(* Schneider Machine Expert - Basic project MIXER_EPP_STARTUP, file version 2.8.0.0 *)
(* CompanyInformations: Name=PROMASS, PhoneNumber=+39074238501, Street=Via XXV Aprile, 10/12, City=Trevi, ZipCode=06039, State=PG, Country=Italy, WebSite=www.promass.com *)
(* ProjectInformations: Name=MIXER_EPP, Description=CONTROL TO MIX-UP RECYCLED EPP (EXANDED POLYPROPILENE) WITH FRESH EPP.
AN ADDITIONAL BLOWE IS ADDED TO PERMIT THE OUTPUT FLOW *)
(* UserInformations: LastName=Torroni, FirstName=Stefano, PhoneNumber=+390742385051, Email=info@promass.com *)

HARDWARE
  Cpu 0: TM221CE16T
  EthernetConfiguration: NetworkName=M221, IpAllocationMode=FixedAddress, IpAddress=192.168.250.10, SubnetMask=255.255.255.0
  SerialLineConfiguration: Baud=Baud19200, Parity=ParityEven, DataBits=DataBits8, StopBits=StopBits1, PhysicalMedium=PhysicalMediumRs485, TransmissionMode=TransmissionModeIoScannerRtu
  MastTask: UsePeriodScanMode=false, PeriodScan=100
  FastTask: Period=255
  CpuBehavior: StartingMode=StartAutoRunForced, AutoSaveRamOnEeprom=true, WatchdogPeriod=250

SYMBOLS  (address, symbol, comment, settings)
  %M0       DRV_PWR_ON
  %M1       DRV0_JOG_INC
  %M2       DRV0_JOG_DEC
  %M3       DRV1_JOG_INC
  %M4       DRV1_JOG_DEC
  %M5       DRV0_MOVE_VEL
  %M6       DRV1_MOVE_VEL
  %M7       DRV0_ERROR
  %M8       DRV1_ERROR
  %M11      UPP_SENS_ON
  %M12      REM_TANK_FULL_V
  %M13      BLOWER_TOF
  %M100     RATIO_0_CHANGED
  %M101     RATIO_1_CHANGED
  %MW0      DRV0_JOG_SPEED
  %MW1      DRV1_JOG_SPEED
  %MW2      DRV0_MOVEVEL_SPEED
  %MW3      DRV1_MOVE_VEL_SPEED
  %MW4      HMI_ALARMS
  %MW5      FSM
  %MW6      HMI_INP  "HMI>>PLC COMMANDS"
  %MW7      HMI_OUT_00  "PLC>>HMI FEEDBACK WORD 01"
  %MW8      HMI_OUT_01  "PLC>>HMI FEEDBACK WORD 02"
  %MW9      SCREW_0_RATIO
  %MW10     SCREW_1_RATIO
  %MW11     BLOWER_DELAY_OFF
  %MW12     UPP_SENS_DELAY_ON
  %MW13     REM_TANK_SENS_DELAY_ON
  %TM11       [Type=TOF, Base=OneSecond, IsDynamicPreset=true]
  %TM13       [Base=OneSecond, IsDynamicPreset=true]
  %MC_JOG_ATV0   [Axis(Value(DriveAxis=DRV0)), Vel(Value(short=30))]
  %MC_JOG_ATV1   [Axis(Value(DriveAxis=DRV1)), Vel(Value(short=15))]
  %MC_MOVEVEL_ATV0   [Axis(Value(DriveAxis=DRV0)), Vel(Value(short=0))]
  %MC_MOVEVEL_ATV1   [Axis(Value(DriveAxis=DRV1)), Vel(Value(short=0))]
  %MC_POWER_ATV0   [Axis(Value(DriveAxis=DRV0))]
  %MC_POWER_ATV1   [Axis(Value(DriveAxis=DRV1))]
  %MC_READMOTIONSTATE_ATV0   [Axis(Value(DriveAxis=DRV0))]
  %MC_READMOTIONSTATE_ATV1   [Axis(Value(DriveAxis=DRV1))]
  %MC_READSTATUS_ATV0   [Axis(Value(DriveAxis=DRV0))]
  %MC_READSTATUS_ATV1   [Axis(Value(DriveAxis=DRV1))]
  %MC_RESET_ATV0   [Axis(Value(DriveAxis=DRV0))]
  %MC_RESET_ATV1   [Axis(Value(DriveAxis=DRV1))]
  %MC_STOP_ATV0   [Axis(Value(DriveAxis=DRV0))]
  %MC_STOP_ATV1   [Axis(Value(DriveAxis=DRV1))]
  %I0.0     START_BTN
  %I0.1     STOP_BTN
  %I0.2     I02
  %I0.3     QM1
  %I0.4     QM2
  %I0.5     QM3
  %I0.6     SK3
  %I0.7     MAT_LVL_UP
  %I0.8     REM_TANK_FULL
  %Q0.0     BLOWER

POU MAIN
  (* SectionNumber=1 *)

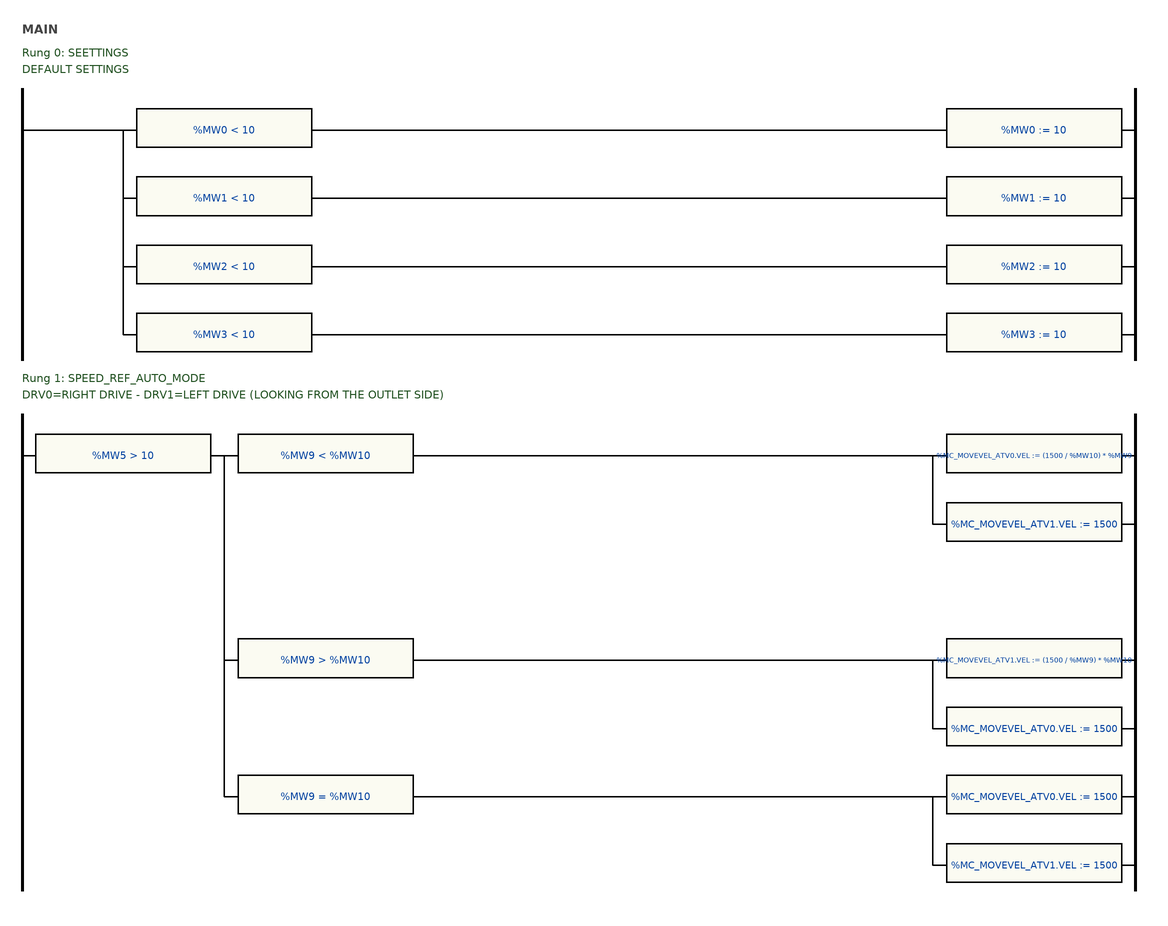

// Rung 0: SEETTINGS
// DEFAULT SETTINGS
  LD 1
  MPS
  AND [ %MW0 < 10 ]       (* DRV0_JOG_SPEED *)
  [ %MW0 := 10 ]          (* DRV0_JOG_SPEED *)
  MRD
  AND [ %MW1 < 10 ]       (* DRV1_JOG_SPEED *)
  [ %MW1 := 10 ]          (* DRV1_JOG_SPEED *)
  MRD
  AND [ %MW2 < 10 ]       (* DRV0_MOVEVEL_SPEED *)
  [ %MW2 := 10 ]          (* DRV0_MOVEVEL_SPEED *)
  MPP
  AND [ %MW3 < 10 ]       (* DRV1_MOVE_VEL_SPEED *)
  [ %MW3 := 10 ]          (* DRV1_MOVE_VEL_SPEED *)
  // as ST:
  //   IF DRV0_JOG_SPEED < 10 THEN DRV0_JOG_SPEED := 10; END_IF;
  //   IF DRV1_JOG_SPEED < 10 THEN DRV1_JOG_SPEED := 10; END_IF;
  //   IF DRV0_MOVEVEL_SPEED < 10 THEN DRV0_MOVEVEL_SPEED := 10; END_IF;
  //   IF DRV1_MOVE_VEL_SPEED < 10 THEN DRV1_MOVE_VEL_SPEED := 10; END_IF;

// Rung 1: SPEED_REF_AUTO_MODE
// DRV0=RIGHT DRIVE - DRV1=LEFT DRIVE (LOOKING FROM THE OUTLET SIDE)
  LD [ %MW5 > 10 ]        (* FSM *)
  MPS
  AND [ %MW9 < %MW10 ]    (* SCREW_0_RATIO, SCREW_1_RATIO *)
  [ %MC_MOVEVEL_ATV0.VEL := ( 1500 / %MW10 ) * %MW9 ](* SCREW_1_RATIO, SCREW_0_RATIO *)
  [ %MC_MOVEVEL_ATV1.VEL := 1500 ]
  MRD
  AND [ %MW9 > %MW10 ]    (* SCREW_0_RATIO, SCREW_1_RATIO *)
  [ %MC_MOVEVEL_ATV1.VEL := ( 1500 / %MW9 ) * %MW10 ](* SCREW_0_RATIO, SCREW_1_RATIO *)
  [ %MC_MOVEVEL_ATV0.VEL := 1500 ]
  MPP
  AND [ %MW9 = %MW10 ]    (* SCREW_0_RATIO, SCREW_1_RATIO *)
  [ %MC_MOVEVEL_ATV0.VEL := 1500 ]
  [ %MC_MOVEVEL_ATV1.VEL := 1500 ]
  // as ST:
  //   IF FSM > 10 AND SCREW_0_RATIO < SCREW_1_RATIO THEN %MC_MOVEVEL_ATV0.VEL := ( 1500 / SCREW_1_RATIO ) * SCREW_0_RATIO; END_IF;
  //   IF FSM > 10 AND SCREW_0_RATIO < SCREW_1_RATIO THEN %MC_MOVEVEL_ATV1.VEL := 1500; END_IF;
  //   IF FSM > 10 AND SCREW_0_RATIO > SCREW_1_RATIO THEN %MC_MOVEVEL_ATV1.VEL := ( 1500 / SCREW_0_RATIO ) * SCREW_1_RATIO; END_IF;
  //   IF FSM > 10 AND SCREW_0_RATIO > SCREW_1_RATIO THEN %MC_MOVEVEL_ATV0.VEL := 1500; END_IF;
  //   IF FSM > 10 AND SCREW_0_RATIO = SCREW_1_RATIO THEN %MC_MOVEVEL_ATV0.VEL := 1500; END_IF;
  //   IF FSM > 10 AND SCREW_0_RATIO = SCREW_1_RATIO THEN %MC_MOVEVEL_ATV1.VEL := 1500; END_IF;

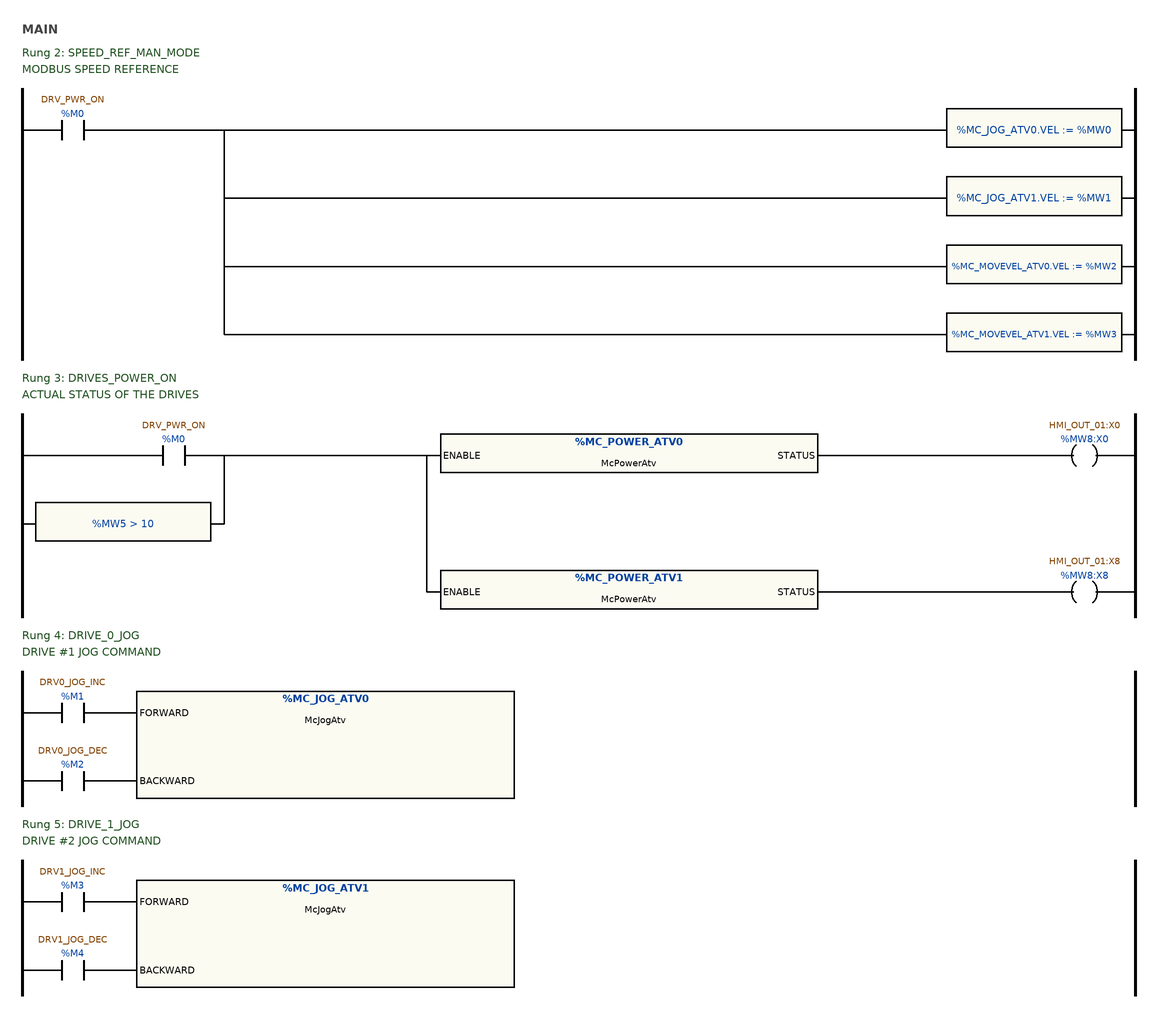

// Rung 2: SPEED_REF_MAN_MODE
// MODBUS SPEED REFERENCE
  LD %M0                  (* DRV_PWR_ON *)
  [ %MC_JOG_ATV0.VEL := %MW0 ](* DRV0_JOG_SPEED *)
  [ %MC_JOG_ATV1.VEL := %MW1 ](* DRV1_JOG_SPEED *)
  [ %MC_MOVEVEL_ATV0.VEL := %MW2 ](* DRV0_MOVEVEL_SPEED *)
  [ %MC_MOVEVEL_ATV1.VEL := %MW3 ](* DRV1_MOVE_VEL_SPEED *)
  // as ST:
  //   IF DRV_PWR_ON THEN %MC_JOG_ATV0.VEL := DRV0_JOG_SPEED; END_IF;
  //   IF DRV_PWR_ON THEN %MC_JOG_ATV1.VEL := DRV1_JOG_SPEED; END_IF;
  //   IF DRV_PWR_ON THEN %MC_MOVEVEL_ATV0.VEL := DRV0_MOVEVEL_SPEED; END_IF;
  //   IF DRV_PWR_ON THEN %MC_MOVEVEL_ATV1.VEL := DRV1_MOVE_VEL_SPEED; END_IF;

// Rung 3: DRIVES_POWER_ON
// ACTUAL STATUS OF THE DRIVES
  LD 1
  MULTIFB
  LD 1
  AND %M0                 (* DRV_PWR_ON *)
  OR [ %MW5 > 10 ]        (* FSM *)
  ST %MW2009:X0
  BLK %MC_POWER_ATV0
  LD %MW2009:X0
  ENABLE
  OUT_BLK
  LD STATUS
  ST %MW8:X0              (* HMI_OUT_01 *)
  END_BLK
  BLK %MC_POWER_ATV1
  LD %MW2009:X0
  ENABLE
  OUT_BLK
  LD STATUS
  ST %MW8:X8              (* HMI_OUT_01 *)
  END_BLK
  MULTIFB
  // as ST:
  //   %MC_POWER_ATV0(ENABLE := DRV_PWR_ON OR FSM > 10);
  //   HMI_OUT_01:X0 := %MC_POWER_ATV0.STATUS;
  //   %MC_POWER_ATV1(ENABLE := DRV_PWR_ON OR FSM > 10);
  //   HMI_OUT_01:X8 := %MC_POWER_ATV1.STATUS;

// Rung 4: DRIVE_0_JOG
// DRIVE #1 JOG COMMAND
  BLK %MC_JOG_ATV0
  LD %M1                  (* DRV0_JOG_INC *)
  FORWARD
  LD %M2                  (* DRV0_JOG_DEC *)
  BACKWARD
  END_BLK
  // as ST:
  //   %MC_JOG_ATV0(FORWARD := DRV0_JOG_INC, BACKWARD := DRV0_JOG_DEC);

// Rung 5: DRIVE_1_JOG
// DRIVE #2 JOG COMMAND
  BLK %MC_JOG_ATV1
  LD %M3                  (* DRV1_JOG_INC *)
  FORWARD
  LD %M4                  (* DRV1_JOG_DEC *)
  BACKWARD
  END_BLK
  // as ST:
  //   %MC_JOG_ATV1(FORWARD := DRV1_JOG_INC, BACKWARD := DRV1_JOG_DEC);

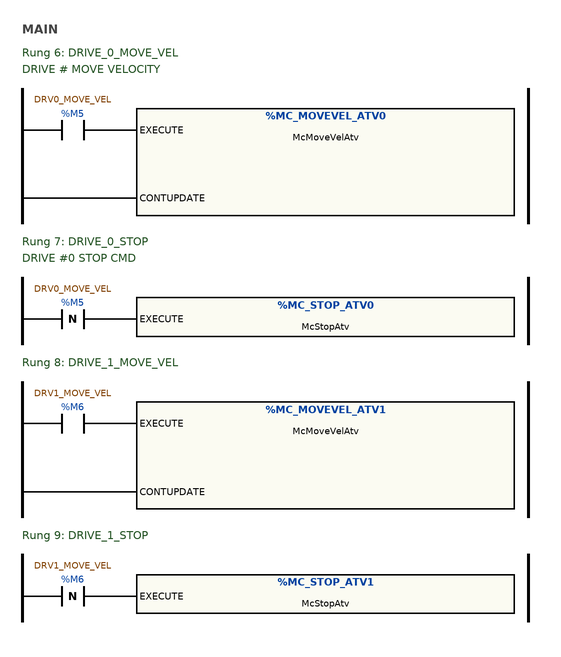

// Rung 6: DRIVE_0_MOVE_VEL
// DRIVE # MOVE VELOCITY
  BLK %MC_MOVEVEL_ATV0
  LD %M5                  (* DRV0_MOVE_VEL *)
  EXECUTE
  LD 1
  CONTUPDATE
  END_BLK
  // as ST:
  //   %MC_MOVEVEL_ATV0(EXECUTE := DRV0_MOVE_VEL, CONTUPDATE := TRUE);

// Rung 7: DRIVE_0_STOP
// DRIVE #0 STOP CMD
  BLK %MC_STOP_ATV0
  LDF %M5                 (* DRV0_MOVE_VEL *)
  EXECUTE
  END_BLK
  // as ST:
  //   %MC_STOP_ATV0(EXECUTE := FALLING(DRV0_MOVE_VEL));

// Rung 8: DRIVE_1_MOVE_VEL
  BLK %MC_MOVEVEL_ATV1
  LD %M6                  (* DRV1_MOVE_VEL *)
  EXECUTE
  LD 1
  CONTUPDATE
  END_BLK
  // as ST:
  //   %MC_MOVEVEL_ATV1(EXECUTE := DRV1_MOVE_VEL, CONTUPDATE := TRUE);

// Rung 9: DRIVE_1_STOP
  BLK %MC_STOP_ATV1
  LDF %M6                 (* DRV1_MOVE_VEL *)
  EXECUTE
  END_BLK
  // as ST:
  //   %MC_STOP_ATV1(EXECUTE := FALLING(DRV1_MOVE_VEL));

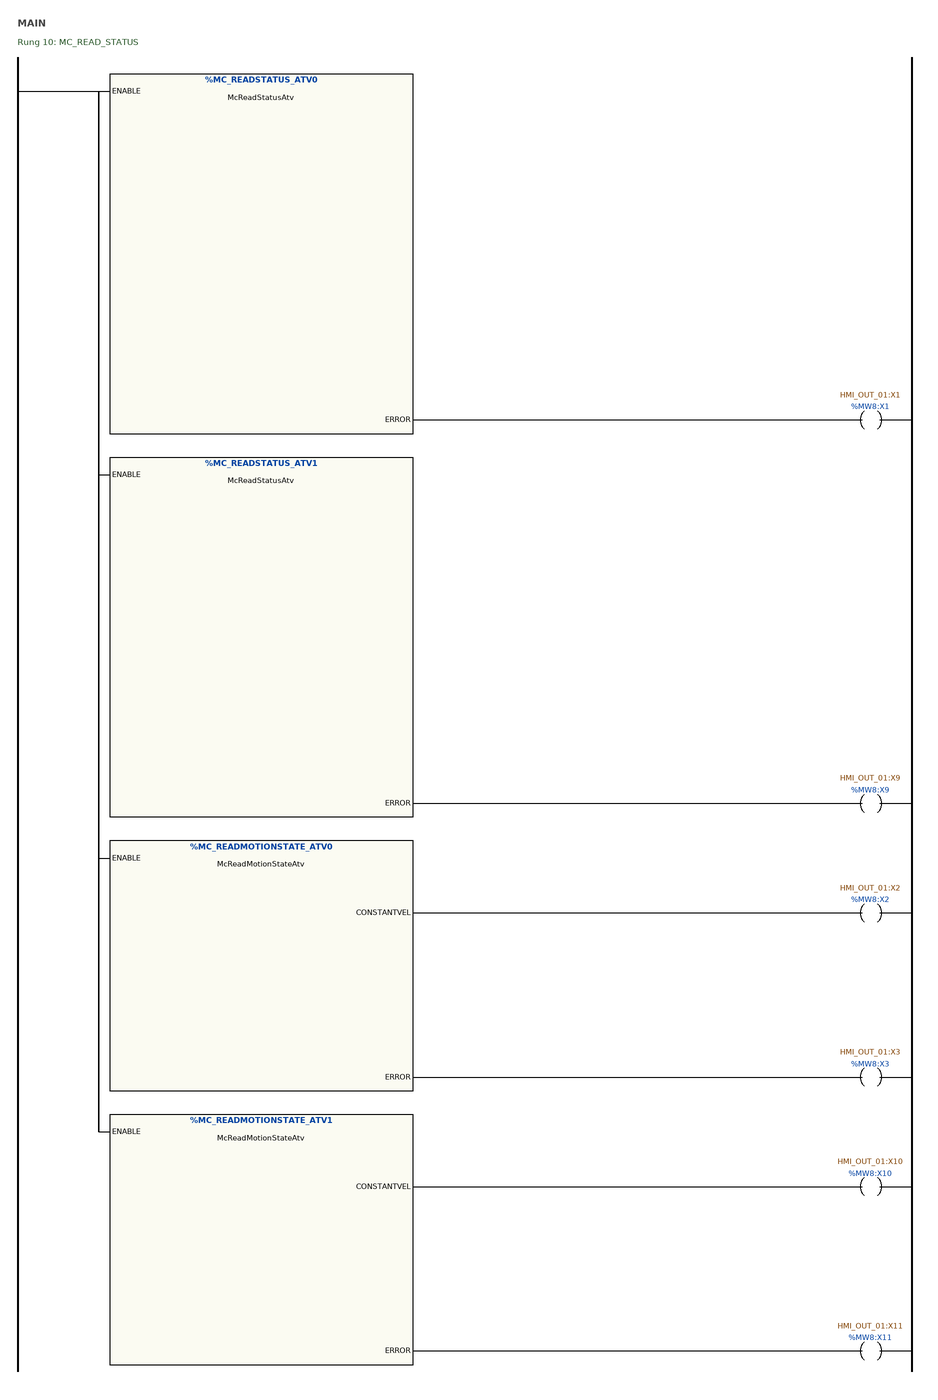

// Rung 10: MC_READ_STATUS
  LD 1
  MULTIFB
  LD 1
  ST %MW2009:X0
  BLK %MC_READSTATUS_ATV0
  LD %MW2009:X0
  ENABLE
  OUT_BLK
  LD ERROR
  ST %MW8:X1              (* HMI_OUT_01 *)
  END_BLK
  BLK %MC_READSTATUS_ATV1
  LD %MW2009:X0
  ENABLE
  OUT_BLK
  LD ERROR
  ST %MW8:X9              (* HMI_OUT_01 *)
  END_BLK
  BLK %MC_READMOTIONSTATE_ATV0
  LD %MW2009:X0
  ENABLE
  OUT_BLK
  LD CONSTANTVEL
  ST %MW8:X2              (* HMI_OUT_01 *)
  LD ERROR
  ST %MW8:X3              (* HMI_OUT_01 *)
  END_BLK
  BLK %MC_READMOTIONSTATE_ATV1
  LD %MW2009:X0
  ENABLE
  OUT_BLK
  LD CONSTANTVEL
  ST %MW8:X10             (* HMI_OUT_01 *)
  LD ERROR
  ST %MW8:X11             (* HMI_OUT_01 *)
  END_BLK
  MULTIFB
  // as ST:
  //   %MC_READSTATUS_ATV0(ENABLE := TRUE);
  //   HMI_OUT_01:X1 := %MC_READSTATUS_ATV0.ERROR;
  //   %MC_READSTATUS_ATV1(ENABLE := TRUE);
  //   HMI_OUT_01:X9 := %MC_READSTATUS_ATV1.ERROR;
  //   %MC_READMOTIONSTATE_ATV0(ENABLE := TRUE);
  //   HMI_OUT_01:X2 := %MC_READMOTIONSTATE_ATV0.CONSTANTVEL;
  //   HMI_OUT_01:X3 := %MC_READMOTIONSTATE_ATV0.ERROR;
  //   %MC_READMOTIONSTATE_ATV1(ENABLE := TRUE);
  //   HMI_OUT_01:X10 := %MC_READMOTIONSTATE_ATV1.CONSTANTVEL;
  //   HMI_OUT_01:X11 := %MC_READMOTIONSTATE_ATV1.ERROR;

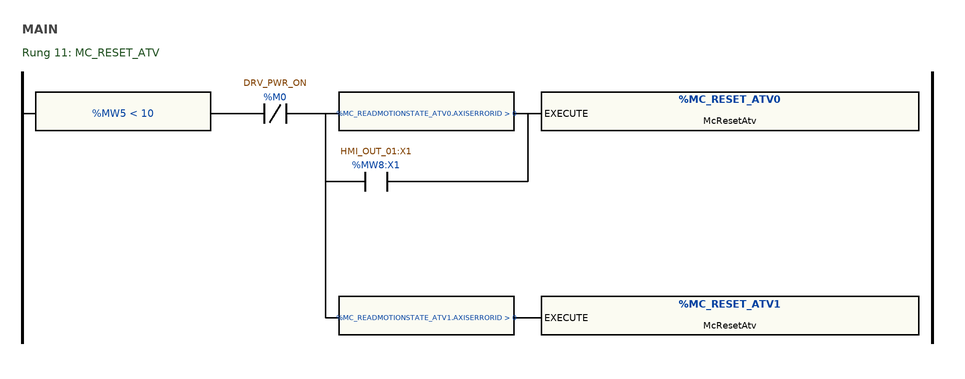

// Rung 11: MC_RESET_ATV
  LD 1
  MULTIFB
  LD 1
  AND [ %MW5 < 10 ]       (* FSM *)
  ANDN %M0                (* DRV_PWR_ON *)
  ST %MW2009:X0
  BLK %MC_RESET_ATV0
  LD %MW2009:X0
  AND( [ %MC_READMOTIONSTATE_ATV0.AXISERRORID > 0 ]
  OR %MW8:X1              (* HMI_OUT_01 *)
  )
  EXECUTE
  END_BLK
  BLK %MC_RESET_ATV1
  LD %MW2009:X0
  AND [ %MC_READMOTIONSTATE_ATV1.AXISERRORID > 0 ]
  EXECUTE
  END_BLK
  MULTIFB
  // as ST:
  //   %MC_RESET_ATV0(EXECUTE := FSM < 10 AND NOT DRV_PWR_ON AND (%MC_READMOTIONSTATE_ATV0.AXISERRORID > 0 OR HMI_OUT_01:X1));
  //   %MC_RESET_ATV1(EXECUTE := FSM < 10 AND NOT DRV_PWR_ON AND %MC_READMOTIONSTATE_ATV1.AXISERRORID > 0);

POU HMI
  (* SectionNumber=2 *)

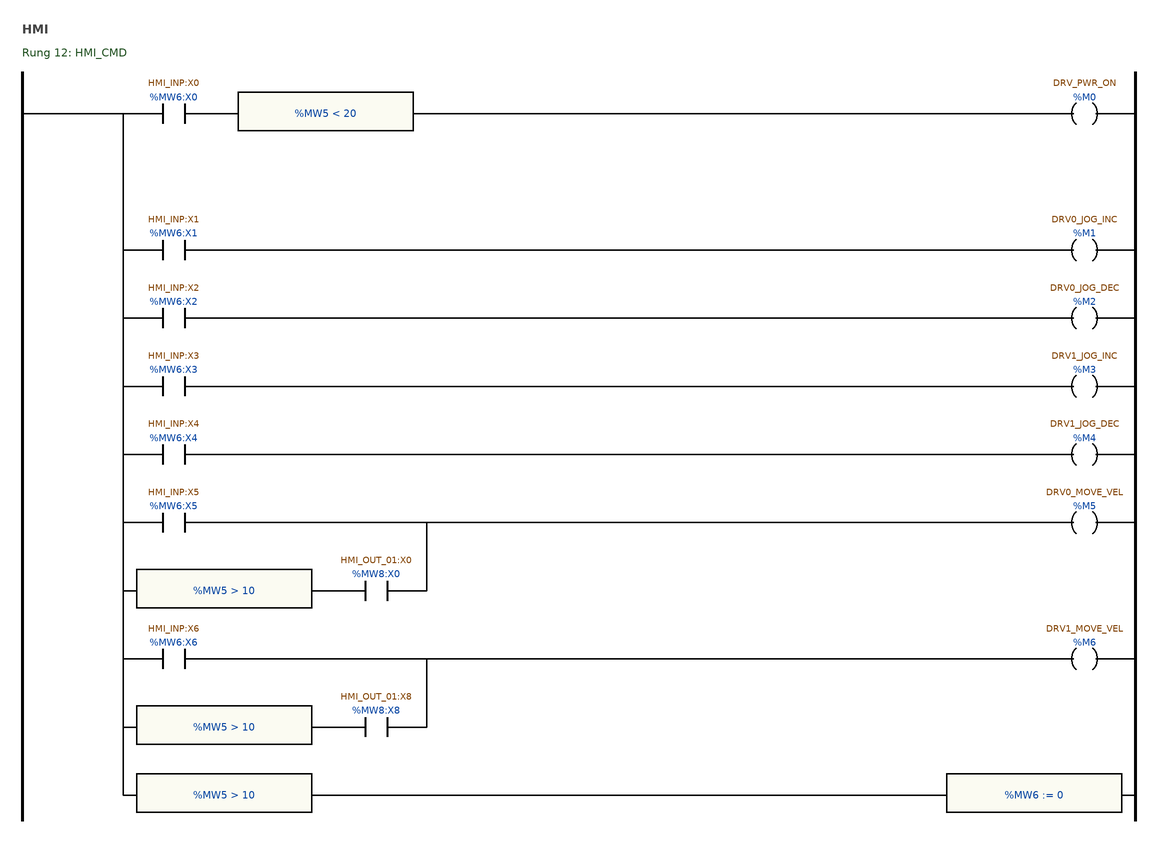

// Rung 12: HMI_CMD
  LD 1
  MPS
  AND %MW6:X0             (* HMI_INP *)
  AND [ %MW5 < 20 ]       (* FSM *)
  ST %M0                  (* DRV_PWR_ON *)
  MRD
  AND %MW6:X1             (* HMI_INP *)
  ST %M1                  (* DRV0_JOG_INC *)
  MRD
  AND %MW6:X2             (* HMI_INP *)
  ST %M2                  (* DRV0_JOG_DEC *)
  MRD
  AND %MW6:X3             (* HMI_INP *)
  ST %M3                  (* DRV1_JOG_INC *)
  MRD
  AND %MW6:X4             (* HMI_INP *)
  ST %M4                  (* DRV1_JOG_DEC *)
  MRD
  AND( %MW6:X5            (* HMI_INP *)
  OR( [ %MW5 > 10 ]       (* FSM *)
  AND %MW8:X0             (* HMI_OUT_01 *)
  )
  )
  ST %M5                  (* DRV0_MOVE_VEL *)
  MRD
  AND( %MW6:X6            (* HMI_INP *)
  OR( [ %MW5 > 10 ]       (* FSM *)
  AND %MW8:X8             (* HMI_OUT_01 *)
  )
  )
  ST %M6                  (* DRV1_MOVE_VEL *)
  MPP
  AND [ %MW5 > 10 ]       (* FSM *)
  [ %MW6 := 0 ]           (* HMI_INP *)
  // as ST:
  //   DRV_PWR_ON := HMI_INP:X0 AND FSM < 20;
  //   DRV0_JOG_INC := HMI_INP:X1;
  //   DRV0_JOG_DEC := HMI_INP:X2;
  //   DRV1_JOG_INC := HMI_INP:X3;
  //   DRV1_JOG_DEC := HMI_INP:X4;
  //   DRV0_MOVE_VEL := HMI_INP:X5 OR FSM > 10 AND HMI_OUT_01:X0;
  //   DRV1_MOVE_VEL := HMI_INP:X6 OR FSM > 10 AND HMI_OUT_01:X8;
  //   IF FSM > 10 THEN HMI_INP := 0; END_IF;

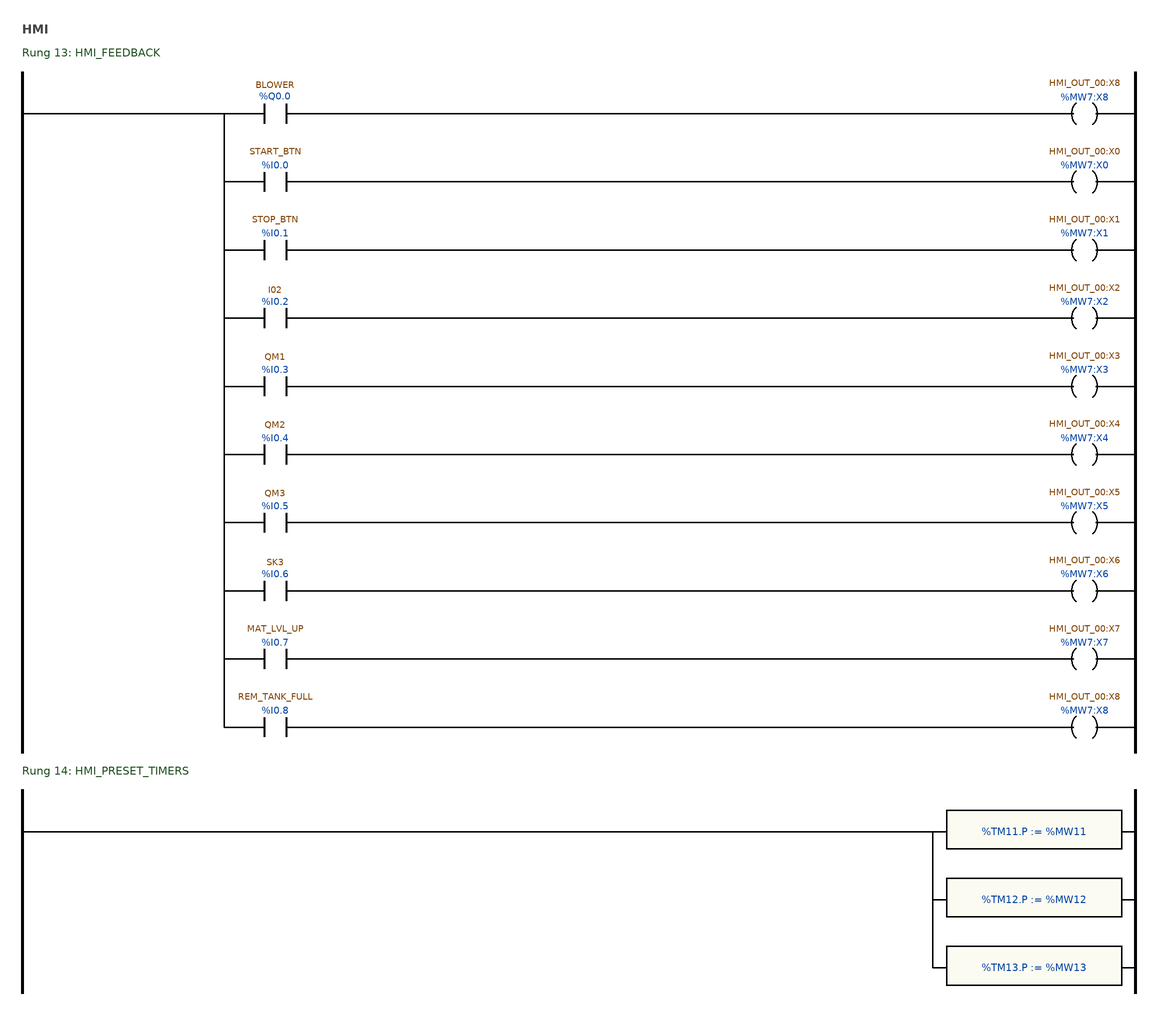

// Rung 13: HMI_FEEDBACK
  LD 1
  MPS
  AND %Q0.0               (* BLOWER *)
  ST %MW7:X8              (* HMI_OUT_00 *)
  MRD
  AND %I0.0               (* START_BTN *)
  ST %MW7:X0              (* HMI_OUT_00 *)
  MRD
  AND %I0.1               (* STOP_BTN *)
  ST %MW7:X1              (* HMI_OUT_00 *)
  MRD
  AND %I0.2               (* I02 *)
  ST %MW7:X2              (* HMI_OUT_00 *)
  MRD
  AND %I0.3               (* QM1 *)
  ST %MW7:X3              (* HMI_OUT_00 *)
  MRD
  AND %I0.4               (* QM2 *)
  ST %MW7:X4              (* HMI_OUT_00 *)
  MRD
  AND %I0.5               (* QM3 *)
  ST %MW7:X5              (* HMI_OUT_00 *)
  MRD
  AND %I0.6               (* SK3 *)
  ST %MW7:X6              (* HMI_OUT_00 *)
  MRD
  AND %I0.7               (* MAT_LVL_UP *)
  ST %MW7:X7              (* HMI_OUT_00 *)
  MPP
  AND %I0.8               (* REM_TANK_FULL *)
  ST %MW7:X8              (* HMI_OUT_00 *)
  // as ST:
  //   HMI_OUT_00:X8 := BLOWER;
  //   HMI_OUT_00:X0 := START_BTN;
  //   HMI_OUT_00:X1 := STOP_BTN;
  //   HMI_OUT_00:X2 := I02;
  //   HMI_OUT_00:X3 := QM1;
  //   HMI_OUT_00:X4 := QM2;
  //   HMI_OUT_00:X5 := QM3;
  //   HMI_OUT_00:X6 := SK3;
  //   HMI_OUT_00:X7 := MAT_LVL_UP;
  //   HMI_OUT_00:X8 := REM_TANK_FULL;

// Rung 14: HMI_PRESET_TIMERS
  LD 1
  [ %TM11.P := %MW11 ]    (* BLOWER_DELAY_OFF *)
  [ %TM12.P := %MW12 ]    (* UPP_SENS_DELAY_ON *)
  [ %TM13.P := %MW13 ]    (* REM_TANK_SENS_DELAY_ON *)
  // as ST:
  //   %TM11.P := BLOWER_DELAY_OFF;
  //   %TM12.P := UPP_SENS_DELAY_ON;
  //   %TM13.P := REM_TANK_SENS_DELAY_ON;

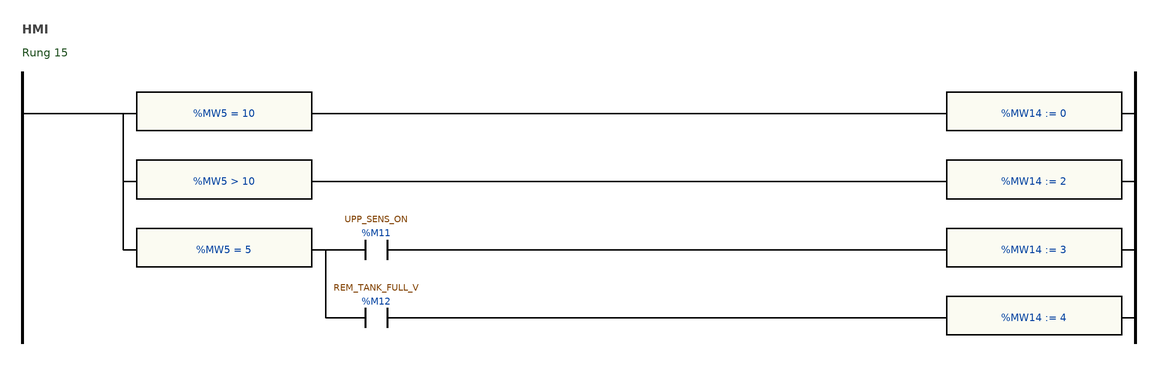

// Rung 15
  LD 1
  MPS
  AND [ %MW5 = 10 ]       (* FSM *)
  [ %MW14 := 0 ]
  MRD
  AND [ %MW5 > 10 ]       (* FSM *)
  [ %MW14 := 2 ]
  MPP
  AND [ %MW5 = 5 ]        (* FSM *)
  MPS
  AND %M11                (* UPP_SENS_ON *)
  [ %MW14 := 3 ]
  MPP
  AND %M12                (* REM_TANK_FULL_V *)
  [ %MW14 := 4 ]
  // as ST:
  //   IF FSM = 10 THEN %MW14 := 0; END_IF;
  //   IF FSM > 10 THEN %MW14 := 2; END_IF;
  //   IF FSM = 5 AND UPP_SENS_ON THEN %MW14 := 3; END_IF;
  //   IF FSM = 5 AND REM_TANK_FULL_V THEN %MW14 := 4; END_IF;

POU FSM
  (* SectionNumber=3 *)

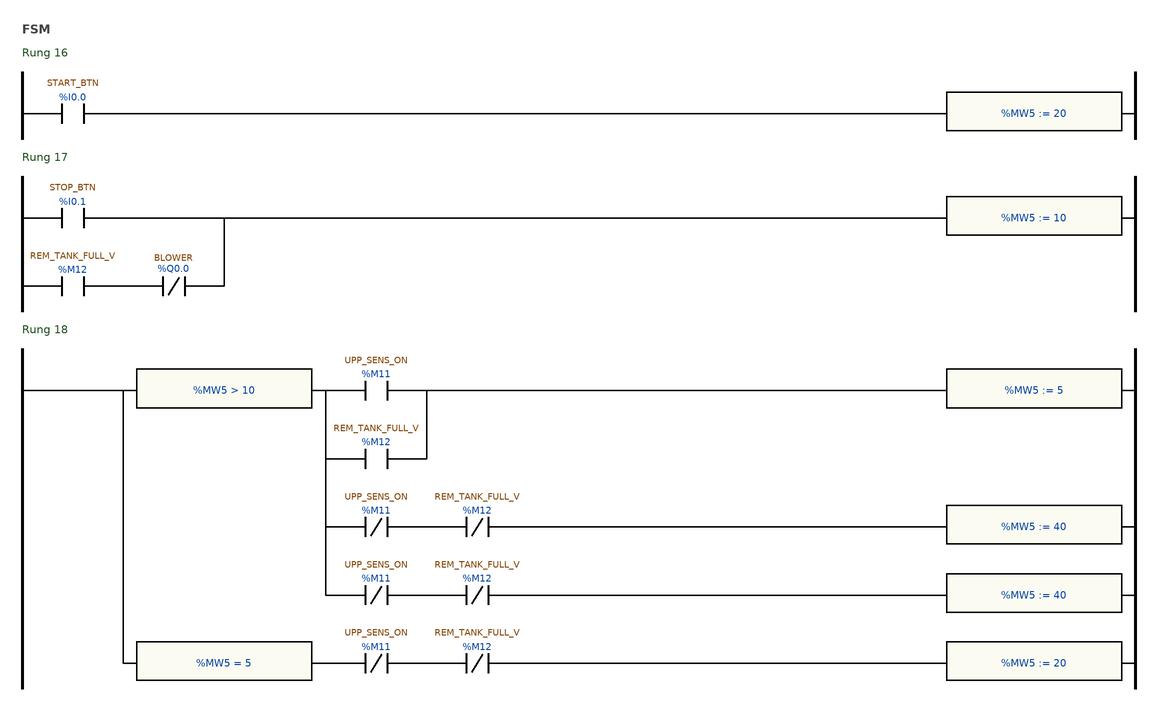

// Rung 16
  LD %I0.0                (* START_BTN *)
  [ %MW5 := 20 ]          (* FSM *)
  // as ST:
  //   IF START_BTN THEN FSM := 20; END_IF;

// Rung 17
  LD %I0.1                (* STOP_BTN *)
  OR( %M12                (* REM_TANK_FULL_V *)
  ANDN %Q0.0              (* BLOWER *)
  )
  [ %MW5 := 10 ]          (* FSM *)
  // as ST:
  //   IF STOP_BTN OR REM_TANK_FULL_V AND NOT BLOWER THEN FSM := 10; END_IF;

// Rung 18
  LD 1
  MPS
  AND [ %MW5 > 10 ]       (* FSM *)
  MPS
  AND( %M11               (* UPP_SENS_ON *)
  OR %M12                 (* REM_TANK_FULL_V *)
  )
  [ %MW5 := 5 ]           (* FSM *)
  MRD
  ANDN %M11               (* UPP_SENS_ON *)
  ANDN %M12               (* REM_TANK_FULL_V *)
  [ %MW5 := 40 ]          (* FSM *)
  MPP
  ANDN %M11               (* UPP_SENS_ON *)
  ANDN %M12               (* REM_TANK_FULL_V *)
  [ %MW5 := 40 ]          (* FSM *)
  MPP
  AND [ %MW5 = 5 ]        (* FSM *)
  ANDN %M11               (* UPP_SENS_ON *)
  ANDN %M12               (* REM_TANK_FULL_V *)
  [ %MW5 := 20 ]          (* FSM *)
  // as ST:
  //   _t1 := FSM > 10;
  //   IF FSM > 10 AND (UPP_SENS_ON OR REM_TANK_FULL_V) THEN FSM := 5; END_IF;
  //   IF _t1 AND NOT UPP_SENS_ON AND NOT REM_TANK_FULL_V THEN FSM := 40; END_IF;
  //   IF _t1 AND NOT UPP_SENS_ON AND NOT REM_TANK_FULL_V THEN FSM := 40; END_IF;
  //   IF FSM = 5 AND NOT UPP_SENS_ON AND NOT REM_TANK_FULL_V THEN FSM := 20; END_IF;

POU TIMERS
  (* SectionNumber=4 *)

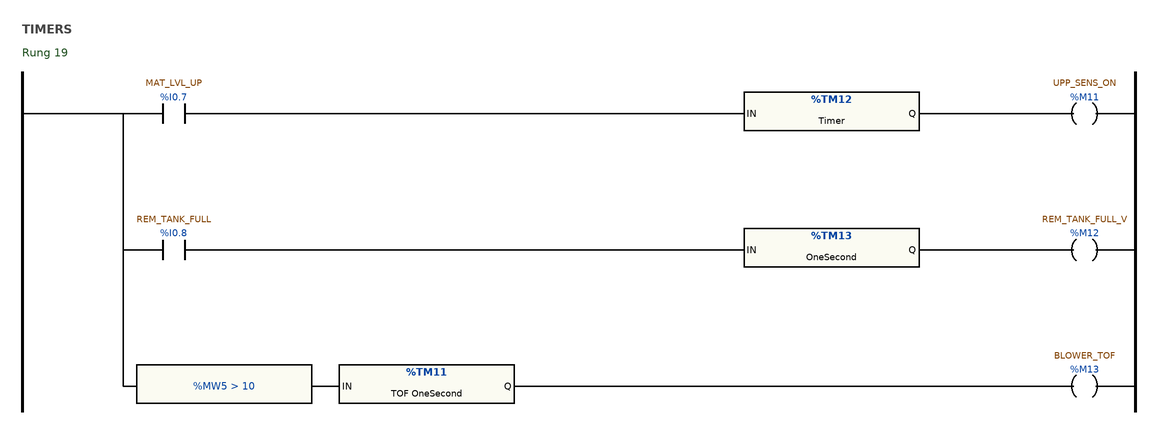

// Rung 19
  LD 1
  MULTIFB
  LD 1
  ST %MW2009:X0
  BLK %TM12
  LD %MW2009:X0
  AND %I0.7               (* MAT_LVL_UP *)
  IN
  OUT_BLK
  LD Q
  ST %M11                 (* UPP_SENS_ON *)
  END_BLK
  BLK %TM13
  LD %MW2009:X0
  AND %I0.8               (* REM_TANK_FULL *)
  IN
  OUT_BLK
  LD Q
  ST %M12                 (* REM_TANK_FULL_V *)
  END_BLK
  BLK %TM11
  LD %MW2009:X0
  AND [ %MW5 > 10 ]       (* FSM *)
  IN
  OUT_BLK
  LD Q
  ST %M13                 (* BLOWER_TOF *)
  END_BLK
  MULTIFB
  // as ST:
  //   %TM12(IN := MAT_LVL_UP);
  //   UPP_SENS_ON := %TM12.Q;
  //   %TM13(IN := REM_TANK_FULL);
  //   REM_TANK_FULL_V := %TM13.Q;
  //   %TM11(IN := FSM > 10);
  //   BLOWER_TOF := %TM11.Q;

POU OUT
  (* SectionNumber=5 *)

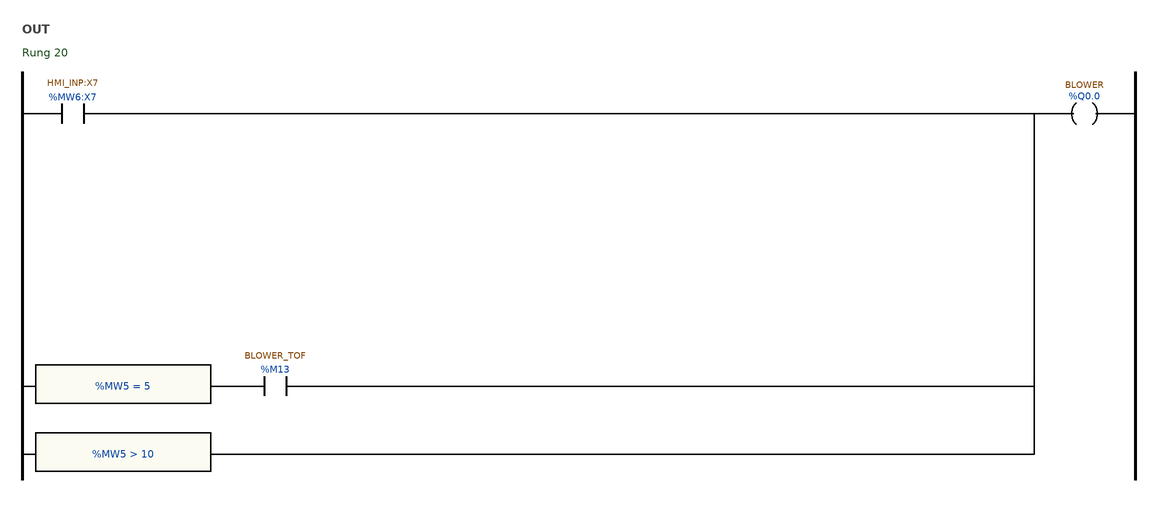

// Rung 20
  LD %MW6:X7              (* HMI_INP *)
  OR( [ %MW5 = 5 ]        (* FSM *)
  AND %M13                (* BLOWER_TOF *)
  )
  OR [ %MW5 > 10 ]        (* FSM *)
  ST %Q0.0                (* BLOWER *)
  // as ST:
  //   BLOWER := HMI_INP:X7 OR FSM = 5 AND BLOWER_TOF OR FSM > 10;

POU RATIO_CALC
  (* SectionNumber=6 *)

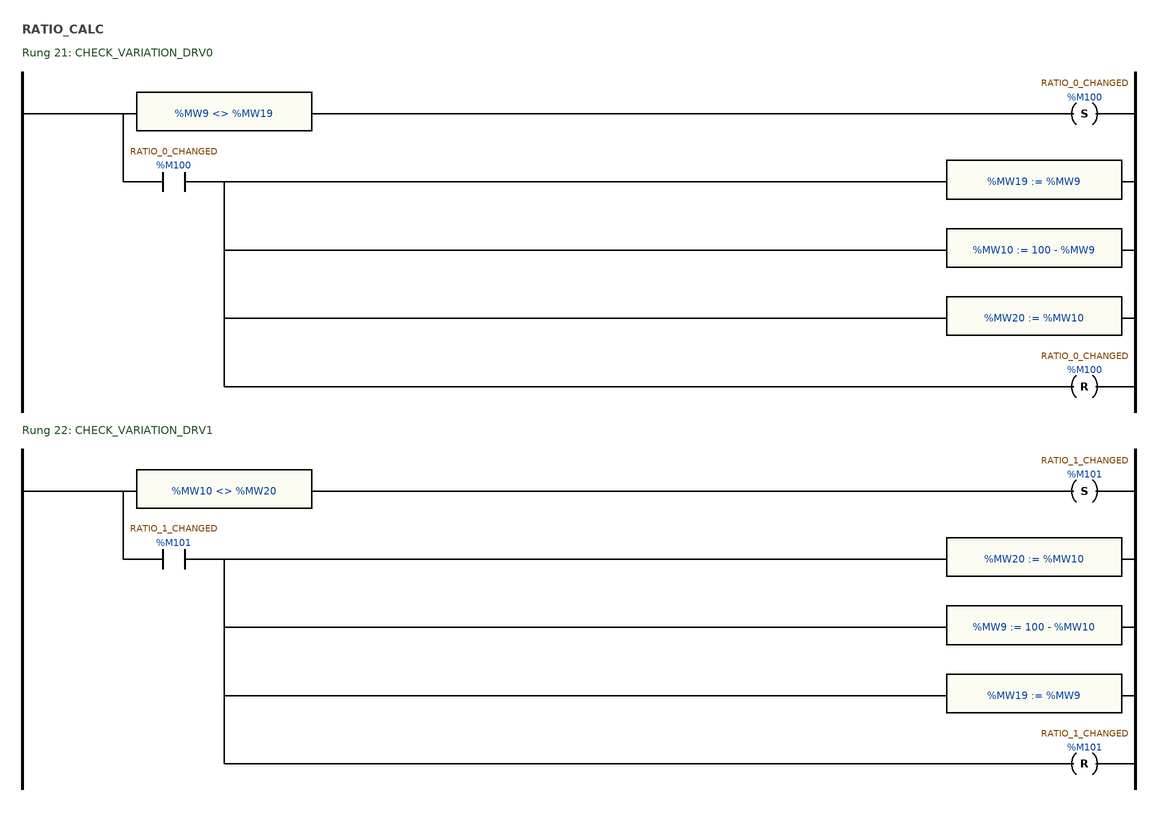

// Rung 21: CHECK_VARIATION_DRV0
  LD 1
  MPS
  AND [ %MW9 <> %MW19 ]   (* SCREW_0_RATIO *)
  S %M100                 (* RATIO_0_CHANGED *)
  MPP
  AND %M100               (* RATIO_0_CHANGED *)
  [ %MW19 := %MW9 ]       (* SCREW_0_RATIO *)
  [ %MW10 := 100 - %MW9 ] (* SCREW_1_RATIO, SCREW_0_RATIO *)
  [ %MW20 := %MW10 ]      (* SCREW_1_RATIO *)
  R %M100                 (* RATIO_0_CHANGED *)
  // as ST:
  //   IF SCREW_0_RATIO <> %MW19 THEN RATIO_0_CHANGED := TRUE; END_IF;
  //   IF RATIO_0_CHANGED THEN %MW19 := SCREW_0_RATIO; END_IF;
  //   IF RATIO_0_CHANGED THEN SCREW_1_RATIO := 100 - SCREW_0_RATIO; END_IF;
  //   IF RATIO_0_CHANGED THEN %MW20 := SCREW_1_RATIO; END_IF;
  //   IF RATIO_0_CHANGED THEN RATIO_0_CHANGED := FALSE; END_IF;

// Rung 22: CHECK_VARIATION_DRV1
  LD 1
  MPS
  AND [ %MW10 <> %MW20 ]  (* SCREW_1_RATIO *)
  S %M101                 (* RATIO_1_CHANGED *)
  MPP
  AND %M101               (* RATIO_1_CHANGED *)
  [ %MW20 := %MW10 ]      (* SCREW_1_RATIO *)
  [ %MW9 := 100 - %MW10 ] (* SCREW_0_RATIO, SCREW_1_RATIO *)
  [ %MW19 := %MW9 ]       (* SCREW_0_RATIO *)
  R %M101                 (* RATIO_1_CHANGED *)
  // as ST:
  //   IF SCREW_1_RATIO <> %MW20 THEN RATIO_1_CHANGED := TRUE; END_IF;
  //   IF RATIO_1_CHANGED THEN %MW20 := SCREW_1_RATIO; END_IF;
  //   IF RATIO_1_CHANGED THEN SCREW_0_RATIO := 100 - SCREW_1_RATIO; END_IF;
  //   IF RATIO_1_CHANGED THEN %MW19 := SCREW_0_RATIO; END_IF;
  //   IF RATIO_1_CHANGED THEN RATIO_1_CHANGED := FALSE; END_IF;
